# EPICS autosave request: iocBoot/gmca_23i_ioc2/dbSave/bluiceHutch.req
$(P)attenuation
